// TIA Portal V16 export
// export: Created 2024-07-31T20:52:03.9780067Z, ExportSetting WithDefaults, DisplayName Totally Integrated Automation Portal, DisplayVersion V16, DisplayName TIA Portal Version Control Interface, DisplayVersion V16, DisplayName TIA Portal Openness, DisplayVersion V16, DisplayName STEP 7 Professional, DisplayVersion V16, DisplayName STEP 7 Safety, DisplayVersion V16, DisplayName WinCC Professional, DisplayVersion V16
VAR_GLOBAL   // PLC tag table "Default tag table"
   START AT %I0.0 : Bool;
   STOP AT %I0.1 : Bool;
   AUTO AT %I0.2 : Bool;
   RESET AT %I0.3 : Bool;
   SORTER_EXTENDED AT %I1.0 : Bool;
   "PARTS_IN _STORAGE" AT %I1.1 : Bool;
   SORTER AT %Q5.0 : Bool;
   CONVEYER AT %Q5.1 : Bool;
END_VAR
